// TIA Portal V19 export
FUNCTION "TONR" : Void   // FC70, STL
TITLE = TIMER ON DELAY - RETENTIVE
{ S7_Optimized_Access := 'TRUE' }
AUTHOR : MODIFIED
FAMILY : TIMERS
NAME : TONR
VERSION : 2.2
// stored: AutoNumber false
   VAR_INPUT
      TMR_EN : Bool;   // Enables timer to accumulate time
      RESET : Bool;   // if = 1, then reset the timer
      PV : DInt;   // Preset value
      DELTA_T : Int;   // OB scan time for previous cycle
   END_VAR
   VAR_OUTPUT
      Q : Bool;   // Set to 1 if timer has timed out
   END_VAR
   VAR_IN_OUT
      ET : DInt;   // Elapsed time
   END_VAR
BEGIN

NETWORK
TITLE = 
// If RESET = 1 then reset the timer by setting Q and ET equal to 0.
      SET;  // RLO := 1
      A     #RESET;  // if(RESET = 1)
      JCN   IF01;  // {
      L     0;  //   ACC1 := 0
      T     #ET;  //   ET := 0
      CLR;  //   RLO := 0
      =     #Q;  //   Q := 0
      JU    EXIT;  // }

// If TMR_EN =1 AND Q =0 then accumulate time by adding DELTA_T to ET. Otherwise, exit function.

IF01: CLR;  // RLO := 0
      L     #ET;  // changed 2/14/00 by ERI per RQ134968
      L     #PV;
      <D;  // IF(ET < PV)
      JCN   EX1;  // {
      CLR;  //   RLO := 0
      O     #TMR_EN;  //   if(TMR_EN = 1)
      JCN   EX1;  //    {
      L     #DELTA_T;  //     ACC1 := DELTA_T
      L     #ET;  //     ACC1 := ET ; ACC2 := DELTA_T
      +D;  //     .
      T     #ET;  //     ET := ET + DELTA_T

// If ET >= PV then set Q = 1, otherwise, exit function

EX1:  L     #ET;  // changed 2/14/00 by ERI per RQ134968
      L     #PV;  //     ACC1 := PV ; ACC2 := ET
      CLR;  //     RLO := 0
      =     #Q;  //     Q := 0
      >=D;  //     IF(ET >= PV)
      JCN   EXIT;  //     {
      SET;  //       RLO := 1
      =     #Q;  //       Q := 1
      NOP   0;  //     }
      NOP   0;  //   }
      NOP   0;  // }

// Exit function successfully by setting the BR bit to a 1.
//
EXIT: SET;  // RLO = 1
      SAVE;  // BR = RLO
END_FUNCTION
